(* IEC 61131-3 sources: JaccoSigma/tempclass/Class/setOuts, 1 file *)

(* ---- setOuts.st ---- *)
(*!
<Class
	Name               = "setOuts"
	Revision           = "0.0"
	RealtimeTask       = "true"
	DefRealtime        = "1 ms"
	CyclicTask         = "false"
	BackgroundTask     = "false"
	Sigmatek           = "false"
	OSInterface        = "false"
	HighPriority       = "false"
	Automatic          = "false"
	UpdateMode         = "Prescan"
	SharedCommandTable = "true"
	Objectsize         = "(284,120)">
	<Channels>
		<Server Name="ClassSvr" Visualized="false" Initialize="false" WriteProtected="false" Retentive="false"/>
		<Server Name="Server" Visualized="false" Initialize="false" WriteProtected="false" Retentive="false"/>
		<Client Name="Client" Required="true" Internal="false"/>
		<Client Name="Client0" Required="true" Internal="false"/>
	</Channels>
</Class>
*)
setOuts : CLASS
  //Servers:
	ClassSvr 	: SvrChCmd_DINT;
	Server 	: SvrCh_UDINT;
  //Clients:
	Client 	: CltCh_DINT;
	Client0 	: CltCh_DINT;
  //Variables:
		Variable 	: UDINT;
  //Functions:

	FUNCTION VIRTUAL GLOBAL RtWork
		VAR_INPUT
			EAX 	: UDINT;
		END_VAR
		VAR_OUTPUT
			state (EAX) 	: UDINT;
		END_VAR;
  //Tables:
	FUNCTION @STD
		VAR_OUTPUT
			ret_code	: CONFSTATES;
		END_VAR;
	FUNCTION GLOBAL TAB @CT_;
END_CLASS;

FUNCTION VIRTUAL GLOBAL setOuts::RtWork
	VAR_INPUT
		EAX 	: UDINT;
	END_VAR
	VAR_OUTPUT
		state (EAX) 	: UDINT;
	END_VAR

  case ClassSvr of
    01:
      Variable := ops.tAbsolute;
      ClassSvr += 1;
      Client.Write(1);
    02:
      if ops.tAbsolute > (Variable+Server) then
        ClassSvr := 99;
        Client0.Write(1);
      end_if;
    00:
      Client.Write(0);
      Client0.Write(0);
  end_case;

	state := READY;

END_FUNCTION
